TYPE PolarisationFilterConfigs :
STRUCT
	FW212CPolarisationFilterConfig : FW212CPolarisationFilterConfig;
	ELL14KPolarisationFilterConfig : ELL14KPolarisationFilterConfig;
END_STRUCT
END_TYPE

(* stored: Version 1.1.0.1, ProductVersion 3.1.4024.3
   DUT PolarisationFilterConfigs: Id {3230fcff-3715-4f4b-963d-6ab306a1ff70} *)
